{region '#Template'}
	{attribute 'Version' := '1.0.0.0'}
	{attribute 'Tags' := '"LCID": "1031", "Text": "Universal, Control, Timer"'}
	{attribute 'Tags' := '"LCID": "1033", "Text": "Universal, Control, Timer"'}
	{attribute 'Description' := '"LCID": "1031", "Text": "Zeitglied Ausschaltverzögert"'}
	{attribute 'Description' := '"LCID": "1033", "Text": "Timer switch-off delayed"'}
{endregion}
FUNCTION_BLOCK FB_BA_DlyOff EXTENDS FB_BA_View
VAR_INPUT
	bVal					: BOOL;	
END_VAR
VAR_OUTPUT
	bQ						: BOOL;	
	nRT						: UDINT;// Restzeit [s] // remaining time [s]
END_VAR
VAR_INPUT CONSTANT
	TiDly					: FB_BA_AV_Op;			
END_VAR	
VAR	
	tofDlyOff				: TOF;
END_VAR
VAR // added by the converter: edge detectors and wires of the graphical bodies
    _w1, _w2 : ANY;
END_VAR

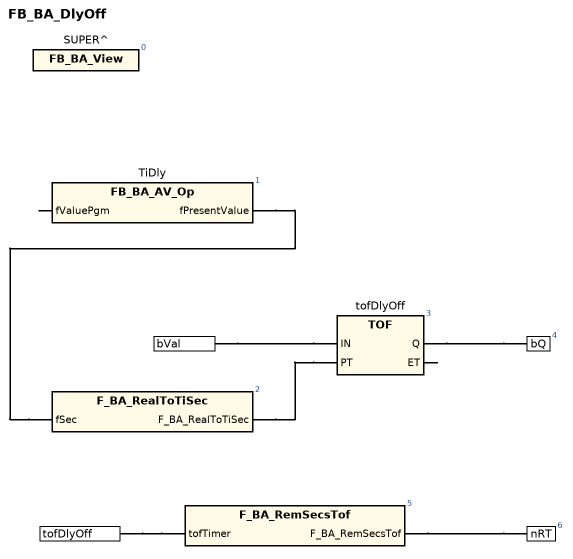
SUPER^(); // FB_BA_View
TiDly(); // FB_BA_AV_Op
_w1 := F_BA_RealToTiSec(fSec := TiDly.fPresentValue);
tofDlyOff(IN := bVal, PT := _w1); // TOF
bQ := tofDlyOff.Q;
_w2 := F_BA_RemSecsTof(tofTimer := tofDlyOff);
nRT := _w2;

METHOD FB_init : BOOL
VAR_INPUT
	bInitRetains : BOOL; // if TRUE, the retain variables are initialized (warm start / cold start)
	bInCopyCode : BOOL;  // if TRUE, the instance afterwards gets moved into the copy code (online change)
END_VAR
TiDly.iParent			:= THIS^;
TiDly.iLabel			:= LblUniControl.DelayOff_TiDly;		 
TiDly.sObjectName		:= '{Idx=01}';								 	 
TiDly.eUnit 			:= E_BA_Unit.eTime_Seconds;								 
TiDly.fValueRm			:= 0;															 
TiDly.fCOVIncrement		:= BA2_Param.fDefCOVIncrement;
END_METHOD

END_FUNCTION_BLOCK

(* stored: Version 1.1.0.1, ProductVersion 3.1.4024.9
   POU FB_BA_DlyOff: Id {a19c0e89-9afd-4e25-82bc-e5741da7617d}, SpecialFunc None
   Method FB_init: Id {ab9caf53-a4a8-4cb0-b4a6-0d6431a5b2dd} *)
